# EPICS autosave request: BPMApp/Db/BPMTrigger_settings.req
$(P)$(R)$(TRIGGER_NAME)$(TRIGGER_CHAN)Chan
$(P)$(R)$(TRIGGER_NAME)$(TRIGGER_CHAN)Dir
$(P)$(R)$(TRIGGER_NAME)$(TRIGGER_CHAN)DirPol
$(P)$(R)$(TRIGGER_NAME)$(TRIGGER_CHAN)RcvLen
$(P)$(R)$(TRIGGER_NAME)$(TRIGGER_CHAN)TrnLen
$(P)$(R)$(TRIGGER_NAME)$(TRIGGER_CHAN)RcvCnt
$(P)$(R)$(TRIGGER_NAME)$(TRIGGER_CHAN)TrnCnt
$(P)$(R)$(TRIGGER_NAME)$(TRIGGER_CHAN)RcvSrc
$(P)$(R)$(TRIGGER_NAME)$(TRIGGER_CHAN)TrnSrc
$(P)$(R)$(TRIGGER_NAME)$(TRIGGER_CHAN)RcvInSel
$(P)$(R)$(TRIGGER_NAME)$(TRIGGER_CHAN)TrnOutSel
